(* Logix 5000 project; controller LAB_5C_MT vendor 1 type 14 code 149 rev 28.12; software revision 28.00 *)

TASK MainTask (continuous, watchdog 500 ms) : MainProgram

MODULES
   Local : vendor 1 type 14 code 149 (Compact 0, rev 28.12)
      Discrete_IO : Embedded (Compact 1, rev 3.1, Output RPI 20 ms)
END_MODULES

PROGRAM MainProgram   (* main routine MainRoutine *)
VAR
   B3_1 : BOOL;   // INTERNAL SHUTDOWN BIT
   IR1 : ALIAS FOR Local:1:I.Data.2;   // COLOR DETECTOR
   IR2 : ALIAS FOR Local:1:I.Data.1;   // METAL DETECTOR
   IR_1 : ALIAS FOR Local:1:I.Data.0;   // PART PRESCENCE
   IR_3 : ALIAS FOR Local:1:I.Data.3;   // PART FINISH
   IR_4 : ALIAS FOR Local:1:O.Data.7;   // PART REQUEST SIGNAL
   LED_1 : ALIAS FOR Local:1:O.Data.8;   // RUN INDICATOR
   LED_2 : ALIAS FOR Local:1:O.Data.9;   // STANDBY INDICATOR
   LED_4 : ALIAS FOR Local:1:O.Data.11;   // Q2 CYCLE STOP
   LED_5 : ALIAS FOR Local:1:O.Data.10;   // Q1 PART REQUEST
   M_1 : ALIAS FOR Local:1:O.Data.0;   // CONVEYOR INDICATOR
   PB_1 : BOOL;   // RESET PBNO PV
   PB_2 : BOOL;   // RUN PBNO
   PB_3 : BOOL := 1;   // STOP PBNC
   PB_4 : BOOL;   // CYCLE STOP
   SOL_1 : ALIAS FOR Local:1:O.Data.1;   // GATE 1
   SOL_2 : ALIAS FOR Local:1:O.Data.2;   // GATE 2
   SOL_3 : ALIAS FOR Local:1:O.Data.4;   // GATE 3
   SOL_4 : ALIAS FOR Local:1:O.Data.3;   // PLUNGER
   SW_1 : BOOL := 1;   // KEY SWITCH PV
   T4_1 : TIMER := (PRE := 1000, ACC := 1000, EN := 1, DN := 1);
END_VAR

ROUTINE MainRoutine   (* ladder *)
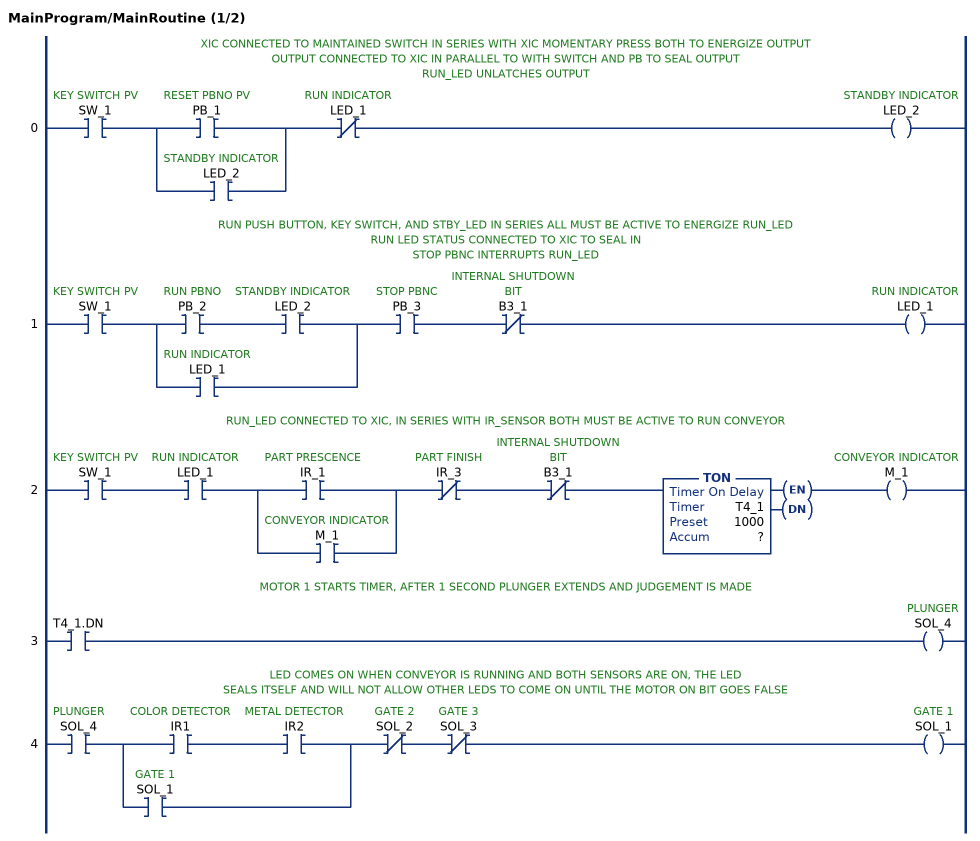
   // XIC CONNECTED TO MAINTAINED SWITCH IN SERIES WITH XIC MOMENTARY PRESS BOTH TO ENERGIZE OUTPUT
   // OUTPUT CONNECTED TO XIC IN PARALLEL TO WITH SWITCH AND PB TO SEAL OUTPUT
   // RUN_LED UNLATCHES OUTPUT
   0: XIC(SW_1)[XIC(PB_1) ,XIC(LED_2) ]XIO(LED_1)OTE(LED_2);
   // RUN PUSH BUTTON, KEY SWITCH, AND STBY_LED IN SERIES ALL MUST BE ACTIVE TO ENERGIZE RUN_LED
   // RUN LED STATUS CONNECTED TO XIC TO SEAL IN
   // STOP PBNC INTERRUPTS RUN_LED
   1: XIC(SW_1)[XIC(PB_2) XIC(LED_2) ,XIC(LED_1) ]XIC(PB_3)XIO(B3_1)OTE(LED_1);
   // RUN_LED CONNECTED TO XIC, IN SERIES WITH IR_SENSOR BOTH MUST BE ACTIVE TO RUN CONVEYOR
   2: XIC(SW_1)XIC(LED_1)[XIC(IR_1) ,XIC(M_1) ]XIO(IR_3)XIO(B3_1)TON(T4_1,?,?)OTE(M_1);
   // MOTOR 1 STARTS TIMER, AFTER 1 SECOND PLUNGER EXTENDS AND JUDGEMENT IS MADE
   3: XIC(T4_1.DN)OTE(SOL_4);
   // LED COMES ON WHEN CONVEYOR IS RUNNING AND BOTH SENSORS ARE ON, THE LED
   // SEALS ITSELF AND WILL NOT ALLOW OTHER LEDS TO COME ON UNTIL THE MOTOR ON BIT GOES FALSE
   4: XIC(SOL_4)[XIC(IR1) XIC(IR2) ,XIC(SOL_1) ]XIO(SOL_2)XIO(SOL_3)OTE(SOL_1);
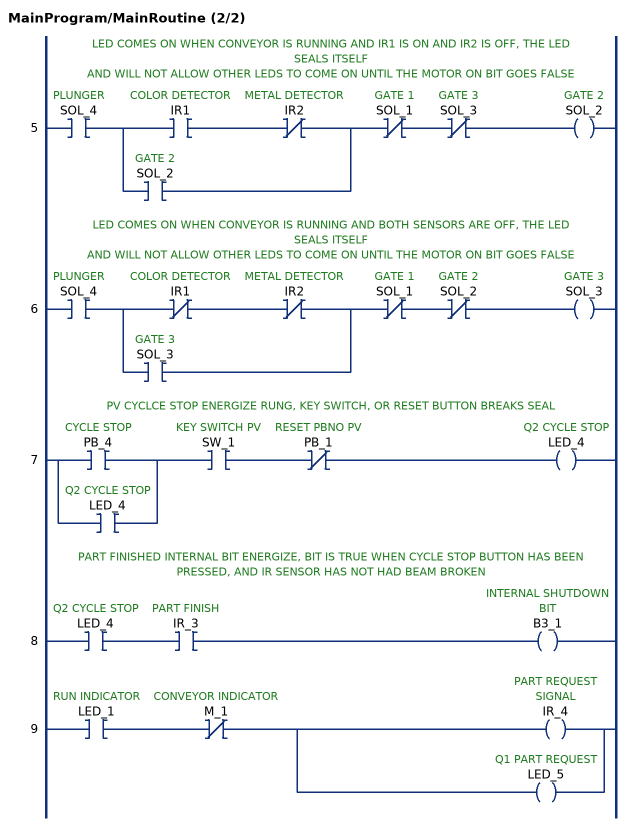
   // LED COMES ON WHEN CONVEYOR IS RUNNING AND IR1 IS ON AND IR2 IS OFF, THE LED SEALS ITSELF
   //  AND WILL NOT ALLOW OTHER LEDS TO COME ON UNTIL THE MOTOR ON BIT GOES FALSE
   5: XIC(SOL_4)[XIC(IR1) XIO(IR2) ,XIC(SOL_2) ]XIO(SOL_1)XIO(SOL_3)OTE(SOL_2);
   // LED COMES ON WHEN CONVEYOR IS RUNNING AND BOTH SENSORS ARE OFF, THE LED SEALS ITSELF
   //  AND WILL NOT ALLOW OTHER LEDS TO COME ON UNTIL THE MOTOR ON BIT GOES FALSE
   6: XIC(SOL_4)[XIO(IR1) XIO(IR2) ,XIC(SOL_3) ]XIO(SOL_1)XIO(SOL_2)OTE(SOL_3);
   // PV CYCLCE STOP ENERGIZE RUNG, KEY SWITCH, OR RESET BUTTON BREAKS SEAL
   7: [XIC(PB_4) ,XIC(LED_4) ]XIC(SW_1)XIO(PB_1)OTE(LED_4);
   // PART FINISHED INTERNAL BIT ENERGIZE, BIT IS TRUE WHEN CYCLE STOP BUTTON HAS BEEN PRESSED, AND IR SENSOR HAS NOT HAD BEAM BROKEN
   8: XIC(LED_4)XIC(IR_3)OTE(B3_1);
   9: XIC(LED_1)XIO(M_1)[OTE(IR_4) ,OTE(LED_5) ];
END_ROUTINE
END_PROGRAM
